FUNCTION_BLOCK PUBLIC FB_Controller
VAR
	fbLampOnOff			:	FB_LampOnOff();
	fbLampSetDirect		:	FB_LampSetDirect();
	fbLampUpDown		:	FB_LampUpDown();
	fbActualValue		:	FB_AnalogValue();
	_eActiveLamp		:	E_LampType;
END_VAR

// Reduces the control value by 5 in the range of 10 to 100. 
METHOD PUBLIC DimDown
CASE _eActiveLamp OF
	E_LampType.OnOff:
		fbLampOnOff.Off();
	E_LampType.SetDirect:
		IF (fbActualValue.nValue >= 15) THEN
			fbLampSetDirect.SetLightLevel(fbActualValue.nValue - 5);
		END_IF
	E_LampType.UpDown:
		IF (fbActualValue.nValue >= 15) THEN
			fbLampUpDown.OneStepDown();
			fbLampUpDown.OneStepDown();
			fbLampUpDown.OneStepDown();
			fbLampUpDown.OneStepDown();
			fbLampUpDown.OneStepDown();
		END_IF
END_CASE
END_METHOD

// Increments the control value by 5 in the range of 10 to 100.
METHOD PUBLIC DimUp
CASE _eActiveLamp OF
	E_LampType.OnOff:
		fbLampOnOff.On();
	E_LampType.SetDirect:
		IF (fbActualValue.nValue <= 95) THEN
			fbLampSetDirect.SetLightLevel(fbActualValue.nValue + 5);
		END_IF
	E_LampType.UpDown:
		IF (fbActualValue.nValue <= 95) THEN
			fbLampUpDown.OneStepUp();
			fbLampUpDown.OneStepUp();
			fbLampUpDown.OneStepUp();
			fbLampUpDown.OneStepUp();
			fbLampUpDown.OneStepUp();
		END_IF
END_CASE
END_METHOD

{attribute 'monitoring' := 'variable'}
PROPERTY PUBLIC eActiveLamp : E_LampType
GET
eActiveLamp := _eActiveLamp;
END_GET
SET
Off();

fbLampOnOff.Detach();
fbLampSetDirect.Detach();
fbLampUpDown.Detach();

CASE eActiveLamp OF
	E_LampType.OnOff:
		fbLampOnOff.Attach(fbActualValue);
	E_LampType.SetDirect:
		fbLampSetDirect.Attach(fbActualValue);
	E_LampType.UpDown:
		fbLampUpDown.Attach(fbActualValue);
END_CASE

_eActiveLamp := eActiveLamp;
END_SET
END_PROPERTY

// Sets the control value to 0.
METHOD PUBLIC Off
CASE _eActiveLamp OF
	E_LampType.OnOff:
		fbLampOnOff.Off();
	E_LampType.SetDirect:
		fbLampSetDirect.SetLightLevel(0);
	E_LampType.UpDown:
		IF (fbActualValue.nValue > 0) THEN
			fbLampUpDown.OnOff();
		END_IF
END_CASE
END_METHOD

// Sets the control value to 100.
METHOD PUBLIC On
CASE _eActiveLamp OF
	E_LampType.OnOff:
		fbLampOnOff.On();
	E_LampType.SetDirect:
		fbLampSetDirect.SetLightLevel(100);
	E_LampType.UpDown:
		IF (fbActualValue.nValue = 0) THEN
			fbLampUpDown.OnOff();
		END_IF
END_CASE
END_METHOD

END_FUNCTION_BLOCK

(* stored: Version 1.1.0.1, ProductVersion 3.1.4024.9
   POU FB_Controller: Id {057b5bd1-e33b-44a4-8eb0-93b60ce9e81d}, SpecialFunc None
   Method DimDown: Id {130de151-930d-42fb-84c7-94f9e80ef2d1}
   Method DimUp: Id {6fad7f57-9367-4e6e-ba7a-7dfd0e3aeed8}
   Property eActiveLamp: Id {1d4afd8b-887b-4e45-b31b-09967b3d8176}
   Get Get: Id {56df7f73-4924-448e-b4c7-e72d89e61bdc}
   Set Set: Id {c2933ac7-b8ac-4726-b19a-e96cc3ec572f}
   Method Off: Id {9d5e0538-50dd-4f19-a271-b30075978c0e}
   Method On: Id {89c7d278-6585-48c0-967a-839fca58784f} *)
